// TIA Portal V16 export
// export: Created 2024-12-03T15:41:46.0669075Z, ExportSetting WithReadOnly, DisplayName Totally Integrated Automation Portal, DisplayVersion V16 Update 6, DisplayName TIA Portal Version Control Interface, DisplayVersion V16 Update 2, DisplayName TIA Portal Openness, DisplayVersion V16 Update 6, DisplayName TIA Portal Teamcenter Gateway, DisplayVersion V16, DisplayName SINAMICS Startdrive Advanced, DisplayVersion V16 Update 5, DisplayName SINAMICS Startdrive G130, G150, S120, S150, SINAMICS MV, S210, DisplayVersion V16 Update 5, DisplayName SINAMICS Startdrive G110M, G120, G120C, G120D, G120P, G115D, DisplayVersion V16 Update 5, DisplayName STEP 7 Professional, DisplayVersion V16 Update 6, DisplayName STEP 7 Safety, DisplayVersion V16, DisplayName WinCC Advanced / Unified PC, DisplayVersion V16 Update 6
TYPE "Parcel_Miscs_UDT"
// stored: CreationDate 2022-02-15T10:12:39.5232481Z, InterfaceModifiedDate 2022-02-15T10:12:59.6958978Z, IsConsistent true, LibraryConformanceStatus The object is library-conformant., ModifiedDate 2022-03-12T11:05:26.0870532Z
   STRUCT
      CuttingOk : Bool;
      cuttingErrror : Bool;
      liddingError : Bool;
      NoCut : Bool;
      NoLid : Bool;
   END_STRUCT;
END_TYPE
